FUNCTION_BLOCK ABSTRACT FBA_TrifectaDrive EXTENDS FBA_Drive
VAR
	outerLimit AT %I* : BOOL;
END_VAR
(*
this abstract FB adds a rear limit sensor to FBA_Drive
*)

{attribute 'monitoring':='call'}
PROPERTY AtOuterLimit : BOOL
GET
AtOuterLimit := outerLimit <> limitSensorDefaultState;
END_GET
END_PROPERTY

END_FUNCTION_BLOCK

(* stored: Version 1.1.0.1, ProductVersion 3.1.4024.11
   POU FBA_TrifectaDrive: Id {08a96a6b-7aa7-42d5-885f-b113fded15c0}, SpecialFunc None
   Property AtOuterLimit: Id {8ff4bd27-c7b3-4485-90d6-8aa8efb8ee2f}
   Get Get: Id {c2019893-210f-47ea-a2dc-1cdf9fa59ef7} *)
